INTERFACE I_NodeFactory

METHOD PUBLIC Create : I_Node
END_METHOD

END_INTERFACE

(* stored: Version 1.1.0.1, ProductVersion 3.1.4024.12
   Itf I_NodeFactory: Id {f17dfa9a-d58a-0253-28a9-a9333d414dc7}
   Method Create: Id {7791efde-3f8b-0c4c-15fc-4d13fe1c8d5a} *)
